Fanuc KAREL source: kc00012.KL

-- PROVISIONAL review KL for V940-1; original PC SHA256 3c3990c4f2ec53f66c9238cc7c64653e669fd15c28caad338d96c72a89c8581a
-- Incomplete behavior may be omitted. Consult companion uncertainty JSON. Do not deploy.
PROGRAM KC00012
%NOLOCKGROUP
BEGIN
  -- V9_ZERO_TABLE_METADATA_HINT layout=0002_ascii; no indexed target words; source/name/runtime held
  -- UNRESOLVED_PC offsets 5-51; opcodes 27,22,22,22,22,22,22,22,31
  -- UNRESOLVED_PC offsets 56-60; opcodes 7F
END KC00012
